{attribute 'qualified_only'}
{attribute 'strict'}
TYPE
    eSetPositionMode :
    (
        Absolute := 0,
        Relative := 1
    );
END_TYPE

(* stored: Version 1.1.0.1, ProductVersion 3.1.4024.12
   DUT eSetPositionMode: Id {0709e9b4-61d0-4137-ad06-b5bf526df03e} *)
